// TwinCAT 3 PLC project Plc_Safe
// ProgramVersion: 3.1.4023.0
// libraries:
//   Tc2_Standard, * (Beckhoff Automation GmbH)
//   Tc2_System, * (Beckhoff Automation GmbH)
//   Tc3_Module, * (Beckhoff Automation GmbH)
//   VisuSymbols,3.5.10.0,System
// project tree:
//   / GlobalTextList.TcGTLO, PlcTask.TcTTO, Visualization Manager.TcVMO (not stored)
//   GVLs/ GVL_IO.TcGVL
//   POUs/ Fb_EdgeDetector.TcPOU (not stored), MAIN.TcPOU, PRG_Safe.TcPOU
//   VISUs/ Visualization_Safe.TcVIS
// real-time tasks:
//   TASK PlcTask: cycle T#10ms, priority 20, ADS port 350

CONFIGURATION Plc_Safe
    RESOURCE PLC ON TwinCAT3
        TASK PlcTask(INTERVAL := T#10ms, PRIORITY := 20);
        PROGRAM MAIN WITH PlcTask : MAIN;
    END_RESOURCE
END_CONFIGURATION

// ---- GVLs/GVL_IO.TcGVL
{attribute 'qualified_only'}
VAR_GLOBAL
	DI_BtnYellow	AT %I*	:	BOOL;
	DI_BtnBlue		AT %I*	:	BOOL;
	DO_LampRed		AT %Q*	:	BOOL;
	DO_LampGreen	AT %Q*	:	BOOL;
END_VAR

// ---- POUs/MAIN.TcPOU
PROGRAM MAIN
VAR
END_VAR

PRG_Safe();

END_PROGRAM

// ---- POUs/PRG_Safe.TcPOU
PROGRAM PRG_Safe
VAR
	edgeDetectorBtnYellow	: Fb_EdgeDetector;
	edgeDetectorBtnBlue		: Fb_EdgeDetector;
	programmingDone			: BOOL;
	codeArray				: ARRAY [1..codeDigits] OF BOOL;
	currentIndex			: INT; 
	correctCounter			: INT; 
	timer					: TON;
	
END_VAR
VAR CONSTANT
	lightDuration			: TIME := T#5S;   // (seconds)
	codeDigits				: INT := 4;
END_VAR

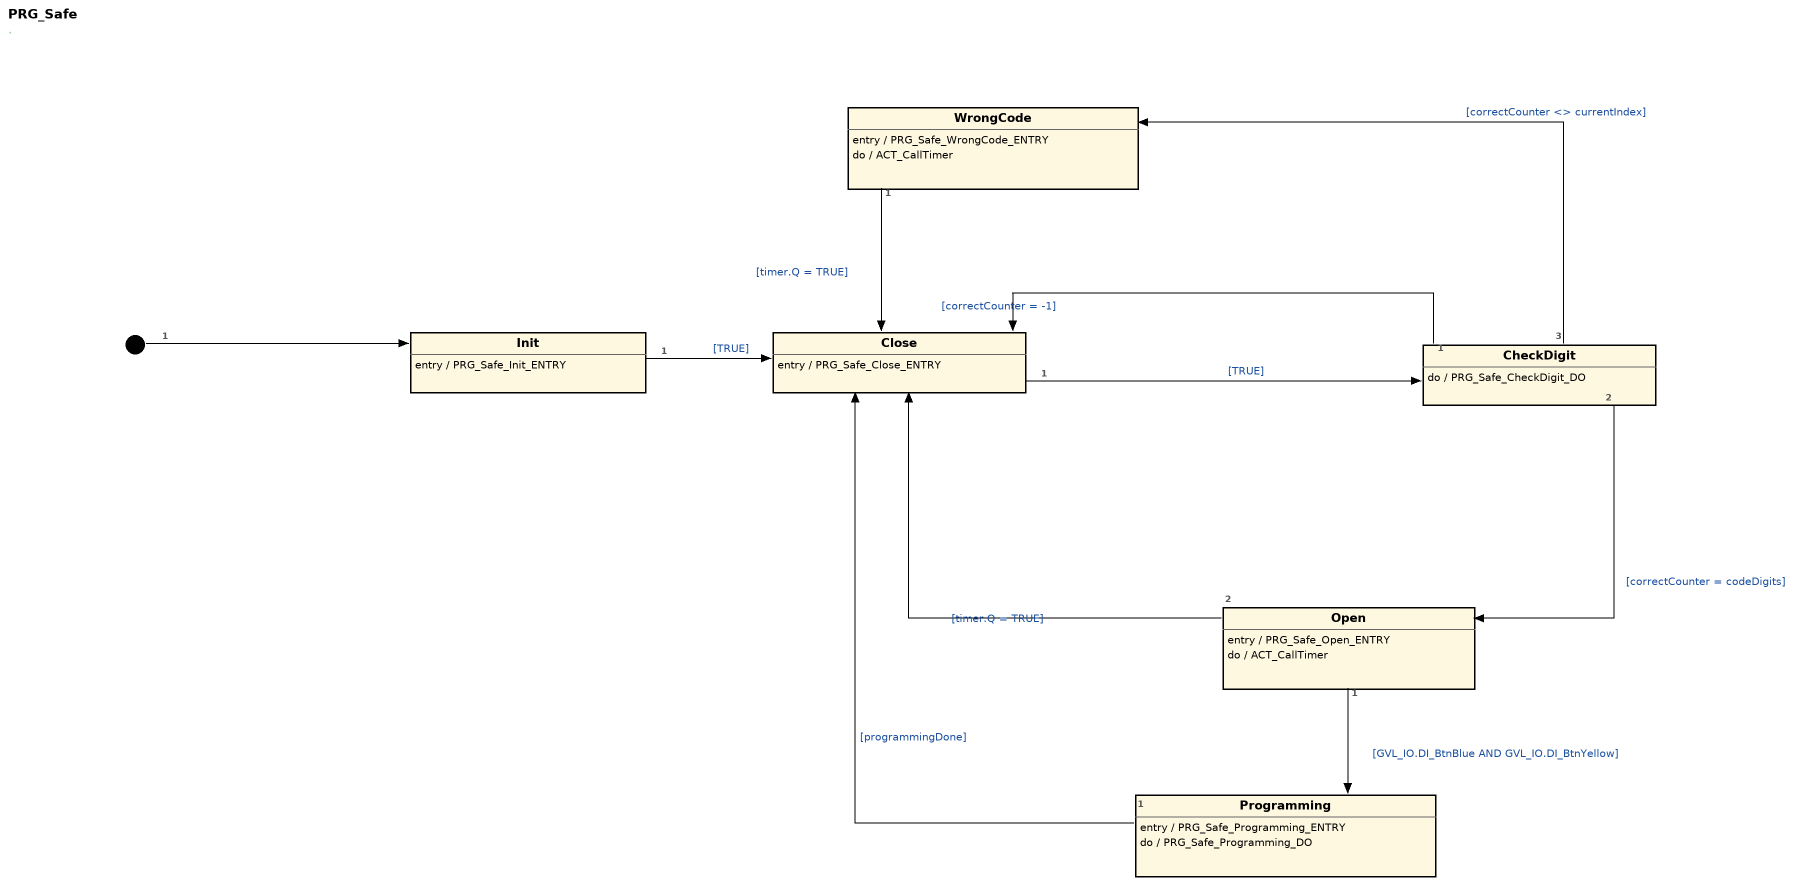
STATECHART PRG_Safe  // abortable
    START StartState1
    NOTEELEMENT 
    STATE WrongCode
        entry / PRG_Safe_WrongCode_ENTRY
        do / ACT_CallTimer
    STATE Init
        entry / PRG_Safe_Init_ENTRY
    STATE Close
        entry / PRG_Safe_Close_ENTRY
    STATE CheckDigit
        do / PRG_Safe_CheckDigit_DO
    STATE Open
        entry / PRG_Safe_Open_ENTRY
        do / ACT_CallTimer
    STATE Programming
        entry / PRG_Safe_Programming_ENTRY
        do / PRG_Safe_Programming_DO
    StartState1 -> Init  // priority 1, on completion
    WrongCode -> Close [timer.Q = TRUE] // priority 1
    Init -> Close [TRUE] // priority 1
    Close -> CheckDigit [TRUE] // priority 1
    CheckDigit -> Close [correctCounter = -1] // priority 1
    CheckDigit -> Open [correctCounter = codeDigits] // priority 2
    CheckDigit -> WrongCode [correctCounter <> currentIndex] // priority 3
    Open -> Programming [GVL_IO.DI_BtnBlue AND GVL_IO.DI_BtnYellow] // priority 1
    Open -> Close [timer.Q = TRUE] // priority 2
    Programming -> Close [programmingDone] // priority 1
END_STATECHART

ACTION ACT_CallTimer:
// call timer function block
timer();
END_ACTION

ACTION PRG_Safe_CheckDigit_DO:
// run edgedetectors
edgeDetectorBtnYellow(inputValue := GVL_IO.DI_BtnYellow);
edgeDetectorBtnBlue(inputValue := GVL_IO.DI_BtnBlue);

// any rising edges?
IF edgeDetectorBtnYellow.risingEdge OR edgeDetectorBtnBlue.risingEdge THEN
	
	// the correct button was pressed
	IF (codeArray[currentIndex+1] = TRUE   AND edgeDetectorBtnYellow.risingEdge) OR
	   (codeArray[currentIndex+1] = FALSE  AND edgeDetectorBtnBlue.risingEdge)   THEN
		correctCounter := correctCounter + 1;
		
	// the wrong button was pressed	
	ELSE
		correctCounter := 0;
	END_IF
	
	currentIndex := currentIndex + 1;
	
END_IF


// double tap blue button
IF edgeDetectorBtnBlue.doublePress THEN
	// will trigger the state change to abort code entry
	correctCounter := -1;
END_IF
END_ACTION

ACTION PRG_Safe_Close_ENTRY:
// reset outputs
GVL_IO.DO_LampGreen := FALSE;
GVL_IO.DO_LampRed := FALSE;

// reset all variables
currentIndex := 0;
correctCounter := 0;
programmingDone := FALSE;

// stop timer
timer.IN := FALSE;
timer();  // call timer so that it resets itself
END_ACTION

ACTION PRG_Safe_Init_ENTRY:
// register correct code
codeArray[1] := TRUE; 
codeArray[2] := FALSE; 
codeArray[3] := TRUE; 
codeArray[4] := FALSE;
END_ACTION

ACTION PRG_Safe_Open_ENTRY:
// light up green lamp
GVL_IO.DO_LampGreen := TRUE;

// configure and start timer
timer.PT := lightDuration;
timer.IN := TRUE;
timer();
END_ACTION

ACTION PRG_Safe_Programming_DO:
// wait until timer is done
timer();
// run edgedetectors
edgeDetectorBtnYellow(inputValue := GVL_IO.DI_BtnYellow);
edgeDetectorBtnBlue(inputValue := GVL_IO.DI_BtnBlue);

IF (timer.Q = FALSE) THEN
	RETURN;
END_IF

// TIMER DONE => proceed

// any rising edges?
IF edgeDetectorBtnYellow.risingEdge OR edgeDetectorBtnBlue.risingEdge THEN
	
	IF edgeDetectorBtnYellow.risingEdge THEN
		codeArray[currentIndex+1] := TRUE;
	ELSIF edgeDetectorBtnBlue.risingEdge THEN
		codeArray[currentIndex+1] := FALSE;
	END_IF
	
	currentIndex := currentIndex + 1;
	
	// finished programming new code
	IF currentIndex = codeDigits THEN
		programmingDone := TRUE;
	END_IF

END_IF
END_ACTION

ACTION PRG_Safe_Programming_ENTRY:
// reset current index
currentIndex := 0;

// signalized programming mode
GVL_IO.DO_LampGreen := TRUE;
GVL_IO.DO_LampRed := TRUE;
timer(IN := FALSE); // reset timer
timer.PT := T#1S;
timer(IN := TRUE); // run timer
END_ACTION

ACTION PRG_Safe_WrongCode_ENTRY:
// light up red lamp
GVL_IO.DO_LampRed := TRUE;

// configure and start timer
timer.PT := lightDuration;
timer.IN := TRUE;
timer();
END_ACTION

END_PROGRAM

// ---- GlobalTextList.TcGTLO
TEXTLIST GlobalTextList
  953 = 'Button '
  429 = 'Code 1'
  329 = 'Code 2'
  874 = 'Code Button 1 (Blue)'
  30 = 'Insert Code:'
  274 = 'Open'
  111 = 'Safe'
  532 = 'Wrong Code'
END_TEXTLIST

// ---- VISUs/Visualization_Safe.TcVIS
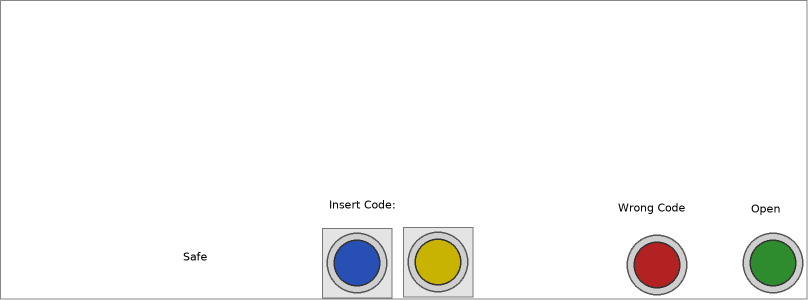
VISUALIZATION Visualization_Safe  // 808x300
    Label (326,190 147x30), "Insert Code:"
    Lamp1 (622,230 70x70), variable: GVL_IO.DO_LampRed, style: Lamp-Lamp1-Red
    PushSwitch (322,228 70x70), variable: GVL_IO.DI_BtnBlue, behaviour: TOGGLE, style: Switch-PushSwitch-Blue
    Lamp1 (738,228 70x70), variable: GVL_IO.DO_LampGreen, style: Lamp-Lamp1-Green
    PushSwitch (403,227 70x70), variable: GVL_IO.DI_BtnYellow, behaviour: TOGGLE, style: Switch-PushSwitch-Yellow
    Label (180,236 59x42), "Safe"
    Label (730,194 72x30), "Open"
    Label (616,193 72x30), "Wrong Code"
END_VISUALIZATION
